PROGRAM PRG_Compilation
VAR
	fbSaMController		: FB_SaMController;
	
END_VAR

END_PROGRAM

(* stored: Version 1.1.0.1
   POU PRG_Compilation: Id {f0171681-5c8e-4bf8-8cd1-9ccd7d95903b}, SpecialFunc None *)
